FUNCTION_BLOCK FB_FigurePlayer
VAR_INPUT
	bStart	: BOOL:= FALSE;
	pFigure : POINTER TO Figure;
	rW_xIn : REAL := 0;
	rW_yIn : REAL := 0;
END_VAR
VAR_OUTPUT
	rW_x : REAL;
	rW_y : REAL;
END_VAR
VAR	
	Visu : ARRAY[0..999] OF VisuElems.VisuStructPoint;
	VisuLenght : INT := 0;
	pVisu : POINTER TO ARRAY[0..999] OF VisuElems.VisuStructPoint;
	counter: UDINT;
END_VAR

IF bStart THEN
	rW_x := pFigure^.X[counter];
	rW_y := pFigure^.Y[counter];
	counter := (counter + 1) MOD pFigure^.length;
ELSE
	rW_x := rW_xIn;
	rW_y := rW_yIn;
	counter := 0;
END_IF

END_FUNCTION_BLOCK

(* stored: Version 1.1.0.1, ProductVersion 3.1.4024.12
   POU FB_FigurePlayer: Id {e03dbe5b-a2fd-4ef6-aba2-1e59fb9a79c7}, SpecialFunc None *)
